TYPE ST_P_CAMERA :
STRUCT
	ProgramName:			STRING;
END_STRUCT
END_TYPE

(* stored: Version 1.1.0.1, ProductVersion 3.1.4024.10
   DUT ST_P_CAMERA: Id {d53cf13b-d8b9-484f-9252-130e91f0e501} *)
